FUNCTION_BLOCK FB_Observable IMPLEMENTS I_Observable
VAR
	_verbose						: BOOL := TRUE;
	// Make sure the list of references to subscribers is updated after online change 
	observers						: ARRAY[0..param.MaxObservers-1] OF I_Observer;
END_VAR

METHOD attach : BOOL
VAR_INPUT
	observer			: I_Observer;
END_VAR
VAR
	i					: INT;
END_VAR
(* default *)
attach := FALSE;

(* loop if the subscriber is already registered *)
FOR i := 0 TO param.MaxObservers-1 DO
	IF observers[i] = observer 	THEN
		observer.update();
		attach := TRUE;
		RETURN;
	END_IF
END_FOR

(* loop for first free position if not yet attached *)
FOR i := 0 TO param.MaxObservers-1 DO
	IF observers[i] = 0 	THEN
		observers[i] := observer;
		message('Observer registered');
		observer.update();
		attach := TRUE;
		EXIT;
	END_IF
END_FOR
END_METHOD

METHOD detach : BOOL
VAR_INPUT
	observer			: I_Observer;
END_VAR
VAR
	i					: INT;
END_VAR
(* default *)
detach := FALSE;

(* loop if the subscriber is already registered *)
FOR i := 0 TO param.MaxObservers-1 DO
	IF observers[i] = observer 	THEN
		observers[i] := 0;
		message('Observer registered');
		detach := TRUE;
		RETURN;
	END_IF
END_FOR
END_METHOD

METHOD INTERNAL message : BOOL
VAR_INPUT
	strArg						: STRING;
END_VAR
// Log message
IF _verbose  THEN
	ADSLOGSTR(
		msgCtrlMask := ADSLOG_MSGTYPE_HINT OR ADSLOG_MSGTYPE_LOG, // ADSLOG_MSGTYPE_ERROR OR ADSLOG_MSGTYPE_LOG, 
		msgFmtStr 	:= '%s',
		strArg 		:= strArg
		);
END_IF
END_METHOD

METHOD notify : BOOL
VAR
	i			: INT;
END_VAR
(* default *)
notify := FALSE;

(* loop if the subscriber is already registered *)
FOR i := 0 TO param.MaxObservers-1 DO
	IF observers[i] <> 0 	THEN
		observers[i].update();
	END_IF
END_FOR
END_METHOD

END_FUNCTION_BLOCK

(* stored: Version 1.1.0.1, ProductVersion 3.1.4024.11
   POU FB_Observable: Id {e2a73847-3ae9-41c4-a05d-e034052bdb33}, SpecialFunc None
   Method attach: Id {8777bfbf-0b24-4d4c-bfbb-b615baf81400}
   Method detach: Id {e9b4dda7-c343-4f9f-a3ca-f5b9e6583823}
   Method message: Id {bdd75991-46b2-4d02-b68d-98ecf52da978}
   Method notify: Id {066cc371-6893-4a9d-a670-ce206a879997} *)
